TYPE PISA_IO :
STRUCT
	sProductName  :STRING;
	bRX AT %I* : BIT;//INPUTS (STATUS -3.4)
	bTX AT %Q* : BIT;//OUTPUTS (CTRL +3.1)
END_STRUCT
END_TYPE

(* stored: Version 1.1.0.1, ProductVersion 3.1.4024.15
   DUT PISA_IO: Id {9d93a83d-6231-4653-afec-ba4fd611ace2} *)
